{attribute addProperty BoxType "EKM1101-0000-0019"}
{attribute addProperty Id "MMS_Device_InputsAT %I*MMS_Device_Inputs_EB48CD741620MMS_Acceleration_StatusAT %I*MMS_Acceleration_Status_2FF1A4723240MMS_Acceleration_X_AxisAT %I*MMS_Acceleration_X_Axis_2EF51F001620MMS_Acceleration_Y_AxisAT %I*MMS_Acceleration_Y_Axis_2EF51F001620MMS_Acceleration_Z_AxisAT %I*MMS_Acceleration_Z_Axis_2EF51F001620MMS_Acceleration_TimestampAT %I*MMS_Acceleration_Timestamp_0B25C1A46480MMS_Voltage_Us_In_InputsAT %I*MMS_Voltage_Us_In_Inputs_BF33E0C16480MMS_Voltage_Up_In_InputsAT %I*MMS_Voltage_Up_In_Inputs_BF33E0C16480MMS_Voltage_Up_Out_InputsAT %I*MMS_Voltage_Up_Out_Inputs_BF33E0C16480MMS_Device_OutputsAT %Q*MMS_Device_Outputs_39C15ABC1620WcStateAT %I*WcState_98A4DF7520.250InfoDataAT %I*InfoData_0BDED7BF144180"}
{attribute addProperty CRC "3393733415"}
{attribute addProperty SizeInBites "514"}
{attribute addProperty SizeInBytes "64.25"}
TYPE EKM1101_87969BFD :
STRUCT
	{attribute addProperty Name "MMS_Device_Inputs"}
	MMS_Device_Inputs : MMS_Device_Inputs_EB48CD74;
	{attribute addProperty Name "MMS_Acceleration_Status"}
	MMS_Acceleration_Status : MMS_Acceleration_Status_2FF1A472;
	{attribute addProperty Name "MMS_Acceleration_X_Axis"}
	MMS_Acceleration_X_Axis : MMS_Acceleration_X_Axis_2EF51F00;
	{attribute addProperty Name "MMS_Acceleration_Y_Axis"}
	MMS_Acceleration_Y_Axis : MMS_Acceleration_Y_Axis_2EF51F00;
	{attribute addProperty Name "MMS_Acceleration_Z_Axis"}
	MMS_Acceleration_Z_Axis : MMS_Acceleration_Z_Axis_2EF51F00;
	{attribute addProperty Name "MMS_Acceleration_Timestamp"}
	MMS_Acceleration_Timestamp : MMS_Acceleration_Timestamp_0B25C1A4;
	{attribute addProperty Name "MMS_Voltage_Us_In_Inputs"}
	MMS_Voltage_Us_In_Inputs : MMS_Voltage_Us_In_Inputs_BF33E0C1;
	{attribute addProperty Name "MMS_Voltage_Up_In_Inputs"}
	MMS_Voltage_Up_In_Inputs : MMS_Voltage_Up_In_Inputs_BF33E0C1;
	{attribute addProperty Name "MMS_Voltage_Up_Out_Inputs"}
	MMS_Voltage_Up_Out_Inputs : MMS_Voltage_Up_Out_Inputs_BF33E0C1;
	{attribute addProperty Name "MMS_Device_Outputs"}
	MMS_Device_Outputs : MMS_Device_Outputs_39C15ABC;
	{attribute addProperty Name "WcState"}
	WcState : WcState_98A4DF75;
	{attribute addProperty Name "InfoData"}
	InfoData : InfoData_0BDED7BF;
END_STRUCT
END_TYPE

(* stored: Version 1.2.0.0, ProductVersion 3.1.4024.9
   DUT EKM1101_87969BFD: Id {db325368-a01f-4292-b060-263c4d652356} *)
